TYPE NCI_REF :
STRUCT
	NCTOPLC_nciref AT %I* : NCTOPLC_NCICHANNEL_REF;
	PLCTONC_nciref AT %Q* : PLCTONC_NCICHANNEL_REF;
END_STRUCT
END_TYPE

(* stored: Version 1.1.0.1, ProductVersion 3.1.4020.3
   DUT NCI_REF: Id {aab8dec0-cc3b-4bc3-8a5f-8144170ac4fb} *)
